// TwinCAT 3 PLC project Untitled1
// ProgramVersion: 3.1.4022.2
// libraries:
//   Tc2_MC2, * (Beckhoff Automation GmbH)
//   Tc2_NC, * (Beckhoff Automation GmbH)
//   Tc2_Standard, * (Beckhoff Automation GmbH)
//   Tc2_System, * (Beckhoff Automation GmbH)
//   Tc3_Module, * (Beckhoff Automation GmbH)
// project tree:
//   GVLs/ Global_Variables.TcGVL
//   / PlcTask.TcTTO
//   POUs/ FB_TcJoy.TcPOU, MAIN.TcPOU
//   POUs/Functions/ MAP.TcPOU
// real-time tasks:
//   TASK PlcTask: cycle T#10ms, priority 20, ADS port 350
// motion (NC):
//   TASK NC-Task 1 SAF: cycle T#2ms, priority 4, ADS port 501
//   TASK NC-Task 1 SVB: cycle T#10ms, priority 8, ADS port 511
//   AXIS Axis 1 (id 1)
//     Dynamic: Acceleration=7107.71, Deceleration=7107.71, Jerk=21323.1
//     Velo: RefSearch=47.3847210666667, RefSync=47.3847210666667, SlowManual=236.923605333333, FastManual=1421.541632, Fast=4738.47210666667, Maximum=4738.47
//     OtherSettings: AllowMotionCmdToSlave=true
//     encoder EncType=8
//       EncPara: ScaleFactorNumerator=104.8576, ScaleFactorDenominator=1048576, MaxCount=#xffffffff
//     drive DrvType=9
//       DrvPara: MaxCount=#xffffffff, DriveControlDWord=#x00030100
//         Analog: VeloReferenz=5212.31931733333, VeloScale=1.02400649589962, ScaleFactorActTorque=0.1
//         TimeComp: TaskDelayCycles=1
//     controller CtrType=1
//       CtrPara: PriorControlFactor=1
//         Observer: BandWidth=20
//   AXIS Axis B (id 2)
//     Dynamic: Acceleration=4539.33952, Deceleration=4539.33952, Jerk=13618.01856
//     Velo: RefSearch=30.2622634666667, RefSync=30.2622634666667, SlowManual=151.311317333333, FastManual=907.867904, Fast=3026.22634666667, Maximum=3026.22634666667
//     OtherSettings: AllowMotionCmdToSlave=true
//     encoder EncType=8
//       EncPara: ScaleFactorNumerator=104.8576, ScaleFactorDenominator=1048576, MaxCount=#xffffffff
//     drive DrvType=9
//       DrvPara: MaxCount=#xffffffff, DriveControlDWord=#x00030100
//         Analog: VeloReferenz=3328.84898133333, VeloScale=1.02400649589962, ScaleFactorActTorque=0.1
//         TimeComp: TaskDelayCycles=1
//     controller CtrType=1
//       CtrPara: PriorControlFactor=1
//         Observer: BandWidth=20
//   AXIS Axis 3 (id 3)
//     OtherSettings: AllowMotionCmdToSlave=true
//     encoder EncType=19
//       EncPara: MaxCount=#xffffffff
//     drive DrvType=16
//       DrvPara: MaxCount=#xffffffff
//         Analog: ScaleFactorActTorque=0.1
//         TimeComp: TaskDelayCycles=1
//     controller CtrType=1
//       CtrPara: PriorControlFactor=1
//         Observer: BandWidth=20
//   AXIS Axis 4 (id 4)
//     Dynamic: Acceleration=167
//     Velo: Maximum=720
//     OtherSettings: AllowMotionCmdToSlave=true
//     encoder EncType=1
//       EncPara: ScaleFactorNumerator=0.005625, Inverse=true
//         Inc: RefSearchInverse=true, RefSyncInverse=false, RefSoftSyncMask=#x0000ffff
//     drive DrvType=24
//       DrvPara: Inverse=true
//         Analog: VeloReferenz=720, ScaleFactorActTorque=0.1
//         TimeComp: TaskDelayCycles=1
//     controller CtrType=1
//       CtrPara: PriorControlFactor=1
//         Observer: BandWidth=20
// I/O:
//   DEVICE Local NIC (EtherCAT), AmsNetId 5.32.241.178.2.1
//     Drive 7 (AX5203-0000-0210) [AX5203-0000-0210 EtherCAT Drive (SoE, 2 Ch.)]
//     Term 1 (EK1100) [EK1100 EtherCAT Coupler (2A E-Bus)]
//       Term 2 (EL3255) [EL3255 5Ch. potentiometer measurement with sensor supply]
//       Term 3 (EL1008) [EL1008 8Ch. Dig. Input 24V, 3ms]
//       Term 4 (EL2008) [EL2008 8Ch. Dig. Output 24V, 0.5A]
//       Term 6 (EL9011) [EL9011 End Terminal]
//     Box 5 (EP2318-0001) [EP2318-0001 4 Ch. Dig. In, 10µs, 4 Ch. Dig. Out 24V, 0,5A, M8]
//   DEVICE Device 2 (EtherCAT), AmsNetId 5.32.241.178.3.1
//     Term 1 (EK1200) [EK1200-5000 EtherCAT Power supply (2A E-Bus)]
//       Term 9 (EL7201-0010) [EL7201-0010 1Ch. MDP742 Servo motor output stage with OCT (50V, 4A)]
//       Term 10 (EL7041) [EL7041 1Ch. Stepper motor output stage (50V, 5A)]
//       Term 4 (EL9011) [EL9011 End Terminal]
// variable links:
//   NC-Task 1 SAF/Axes/Axis 1 <-> Local NIC (EtherCAT)/Drive 7 (AX5203-0000-0210)
//     Drive/Inputs/In/nDataIn1 <-> AT 1/Following distance
//     Drive/Inputs/In/nDcOutputTime <-> InfoData/DcOutputShift
//     Drive/Inputs/In/nState1 <-> AT 1/Drive status word @bit 8
//     Drive/Inputs/In/nState2 <-> AT 1/Drive status word
//     Drive/Inputs/In/nState4 @bit 1 <-> WcState/InputToggle
//     Drive/Inputs/In/nState4 <-> WcState/WcState
//     Drive/Outputs/Out/nCtrl1 <-> MDT 1/Master control word @bit 8
//     Drive/Outputs/Out/nDataOut1 <-> MDT 1/Position command value
//     Enc/Inputs/In/nDataIn1 <-> AT 1/Position feedback 1 value
//     Enc/Inputs/In/nDcInputTime <-> InfoData/DcInputShift
//     Enc/Inputs/In/nState4 @bit 1 <-> WcState/InputToggle
//     Enc/Inputs/In/nState4 <-> WcState/WcState
//   NC-Task 1 SAF/Axes/Axis 3 <-> Device 2 (EtherCAT)/Term 1 (EK1200)/Term 9 (EL7201-0010)
//     Drive/Inputs/In/nDcOutputTime <-> InfoData/DcOutputShift
//     Drive/Inputs/In/nState1 <-> DRV Statusword/Statusword
//     Drive/Inputs/In/nState2 <-> DRV Statusword/Statusword @bit 8
//     Drive/Inputs/In/nState4 @bit 1 <-> WcState/InputToggle
//     Drive/Inputs/In/nState4 <-> WcState/WcState
//     Drive/Outputs/Out/nCtrl1 <-> DRV Controlword/Controlword
//     Drive/Outputs/Out/nCtrl2 <-> DRV Controlword/Controlword @bit 8
//     Drive/Outputs/Out/nDataOut2 <-> DRV Target velocity/Target velocity
//     Enc/Inputs/In/nDataIn1 <-> FB Position/Position
//     Enc/Inputs/In/nDcInputTime <-> InfoData/DcInputShift
//     Enc/Inputs/In/nState4 @bit 1 <-> WcState/InputToggle
//     Enc/Inputs/In/nState4 <-> WcState/WcState
//   NC-Task 1 SAF/Axes/Axis 4 <-> Device 2 (EtherCAT)/Term 1 (EK1200)/Term 10 (EL7041)
//     Drive/Inputs/In/nState1 @bit 3 <-> STM Status/Status/Error
//     Drive/Inputs/In/nState1 @bit 5 <-> STM Status/Status/Moving negative
//     Drive/Inputs/In/nState1 @bit 4 <-> STM Status/Status/Moving positive
//     Drive/Inputs/In/nState1 @bit 1 <-> STM Status/Status/Ready
//     Drive/Inputs/In/nState1 <-> STM Status/Status/Ready to enable
//     Drive/Inputs/In/nState1 @bit 6 <-> STM Status/Status/Torque reduced
//     Drive/Inputs/In/nState1 @bit 2 <-> STM Status/Status/Warning
//     Drive/Inputs/In/nState2 @bit 3 <-> STM Status/Status/Digital input 1
//     Drive/Inputs/In/nState2 @bit 4 <-> STM Status/Status/Digital input 2
//     Drive/Inputs/In/nState2 @bit 5 <-> STM Status/Status/Sync error
//     Drive/Inputs/In/nState2 @bit 7 <-> STM Status/Status/TxPDO Toggle
//     Drive/Inputs/In/nState4 @bit 1 <-> WcState/InputToggle
//     Drive/Inputs/In/nState4 <-> WcState/WcState
//     Drive/Outputs/Out/nCtrl1 <-> STM Control/Control/Enable
//     Drive/Outputs/Out/nCtrl1 @bit 2 <-> STM Control/Control/Reduce torque
//     Drive/Outputs/Out/nCtrl1 @bit 1 <-> STM Control/Control/Reset
//     Drive/Outputs/Out/nDataOut2[0] <-> STM Velocity/Velocity
//     Enc/Inputs/In/nDataIn1[0] <-> ENC Status compact/Counter value
//     Enc/Inputs/In/nDataIn2[0] <-> ENC Status compact/Latch value
//     Enc/Inputs/In/nState1 @bit 4 <-> ENC Status compact/Status/Counter overflow
//     Enc/Inputs/In/nState1 @bit 3 <-> ENC Status compact/Status/Counter underflow
//     Enc/Inputs/In/nState1 @bit 7 <-> ENC Status compact/Status/Extrapolation stall
//     Enc/Inputs/In/nState1 <-> ENC Status compact/Status/Latch C valid
//     Enc/Inputs/In/nState1 @bit 1 <-> ENC Status compact/Status/Latch extern valid
//     Enc/Inputs/In/nState1 @bit 2 <-> ENC Status compact/Status/Set counter done
//     Enc/Inputs/In/nState2 @bit 4 <-> ENC Status compact/Status/Status of extern latch
//     Enc/Inputs/In/nState2 <-> ENC Status compact/Status/Status of input A
//     Enc/Inputs/In/nState2 @bit 1 <-> ENC Status compact/Status/Status of input B
//     Enc/Inputs/In/nState2 @bit 2 <-> ENC Status compact/Status/Status of input C
//     Enc/Inputs/In/nState2 @bit 5 <-> ENC Status compact/Status/Sync error
//     Enc/Inputs/In/nState2 @bit 7 <-> ENC Status compact/Status/TxPDO Toggle
//     Enc/Inputs/In/nState4 @bit 1 <-> WcState/InputToggle
//     Enc/Inputs/In/nState4 <-> WcState/WcState
//     Enc/Outputs/Out/nCtrl1 <-> ENC Control compact/Control/Enable latch C
//     Enc/Outputs/Out/nCtrl1 @bit 3 <-> ENC Control compact/Control/Enable latch extern on negative edge
//     Enc/Outputs/Out/nCtrl1 @bit 1 <-> ENC Control compact/Control/Enable latch extern on positive edge
//     Enc/Outputs/Out/nCtrl1 @bit 2 <-> ENC Control compact/Control/Set counter
//     Enc/Outputs/Out/nDataOut1[0] <-> ENC Control compact/Set counter value
//   NC-Task 1 SAF/Axes/Axis B <-> Local NIC (EtherCAT)/Drive 7 (AX5203-0000-0210)
//     Drive/Inputs/In/nDataIn1 <-> AT 2/Following distance
//     Drive/Inputs/In/nDcOutputTime <-> InfoData/DcOutputShift
//     Drive/Inputs/In/nState1 <-> AT 2/Drive status word @bit 8
//     Drive/Inputs/In/nState2 <-> AT 2/Drive status word
//     Drive/Inputs/In/nState4 @bit 1 <-> WcState/InputToggle
//     Drive/Inputs/In/nState4 <-> WcState/WcState
//     Drive/Outputs/Out/nCtrl1 <-> MDT 2/Master control word @bit 8
//     Drive/Outputs/Out/nDataOut1 <-> MDT 2/Position command value
//     Enc/Inputs/In/nDataIn1 <-> AT 2/Position feedback 1 value
//     Enc/Inputs/In/nDcInputTime <-> InfoData/DcInputShift
//     Enc/Inputs/In/nState4 @bit 1 <-> WcState/InputToggle
//     Enc/Inputs/In/nState4 <-> WcState/WcState
//   Untitled1/Untitled1 Instance <-> Local NIC (EtherCAT)/Term 1 (EK1100)/Term 2 (EL3255)
//     PlcTask Inputs/MAIN.Throttle <-> AI Standard Channel 1/Value
//   Untitled1/Untitled1 Instance <-> Local NIC (EtherCAT)/Term 1 (EK1100)/Term 3 (EL1008)
//     PlcTask Inputs/MAIN.prox <-> Channel 5/Input
//   Untitled1/Untitled1 Instance <-> Local NIC (EtherCAT)/Term 1 (EK1100)/Term 4 (EL2008)
//     PlcTask Outputs/MAIN.four <-> Channel 4/Output
//     PlcTask Outputs/MAIN.one <-> Channel 1/Output
//     PlcTask Outputs/MAIN.three <-> Channel 3/Output
//     PlcTask Outputs/MAIN.two <-> Channel 2/Output
//   Untitled1/Untitled1 Instance <-> NC-Task 1 SAF/Axes/Axis 4
//     PlcTask Inputs/MAIN.AxisB.NcToPlc <-> Outputs/ToPlc
//     PlcTask Outputs/MAIN.AxisB.PlcToNc <-> Inputs/FromPlc

CONFIGURATION Untitled1
    RESOURCE PLC ON TwinCAT3
        TASK PlcTask(INTERVAL := T#10ms, PRIORITY := 20);
        PROGRAM MAIN WITH PlcTask : MAIN;
    END_RESOURCE
END_CONFIGURATION

// ---- GVLs/Global_Variables.TcGVL
VAR_GLOBAL
	
END_VAR

// ---- POUs/MAIN.TcPOU
PROGRAM MAIN
VAR
	
    heartbeat : BYTE;
	
	// Outputs.
	one AT %Q* : BOOL;
	two AT %Q* : BOOL;
	three AT %Q* : BOOL;
	four AT %Q* : BOOL;
	
	prox AT %I* : BOOL;  // Input
	
	// Dynamic Throttle
	Throttle AT %I* : INT;
	LastThrottle : INT;
	
	AxisB : AXIS_REF;

	McPower : MC_Power;
	McReset : MC_Reset;
	McJogging : MC_Jog;
	McVelocity : MC_MoveVelocity;
	McStop : MC_Stop;
	McHome : MC_Home;

	
    CurrentVelocityCmd : DINT;

	iState : DINT; // My State

	McMoveAbs : MC_MoveAbsolute;
	McMoveRel : MC_MoveRelative;
	iNumMoves : DINT:= 5;
	iCurrMove : DINT;
	fMoveDistEachTime : REAL:= 10;
	fRelMoveDist : REAL;
	
	TcJoy : FB_TcJoy;

END_VAR

heartbeat := heartbeat + 1;

CurrentVelocityCmd := MAP(Throttle,29800,22600,0,2800);
IF CurrentVelocityCmd < 50 THEN
	CurrentVelocityCmd := 0;
END_IF

AxisB.ReadStatus();

McPower(Axis:=AxisB,Enable:=TRUE,Enable_Positive:=TRUE,Enable_Negative:=TRUE);
McReset(Axis:=AxisB);
McJogging(Axis:=AxisB);
McHome(Axis:=AxisB,bCalibrationCam := prox);

McMoveAbs(Axis:=AxisB);
McMoveRel(Axis:=AxisB);

TcJoy();

CASE iState OF
	
    0:  // Initial

		iState := 10;

    10:  // Start Drive Reset

		McHome(Axis:=AxisB,Execute:=FALSE);
		McReset(Axis:=AxisB,Execute:=TRUE);
		IF McReset.Done THEN
			iState :=20;
		ELSIF McReset.Error THEN
			iState := 999;
		END_IF

    20:  // Wait for Drive to Reset

		IF McPower.Status AND (CurrentVelocityCmd > 1000 OR TcJoy.Y_Button) THEN
			iState := 100;
		END_IF	
		
    30:  // Wait for drive JOG command.
    
		IF TcJoy.iRightTrigger_Axis > 0 THEN
	
			IF TcJoy.iRightStick_X_Axis > 0 THEN
				McJogging.JogForward := TRUE;
				McJogging.Velocity := ABS(MAP(TcJoy.iRightStick_X_Axis,6000,32767,0,720));
			ELSE
				McJogging.JogForward := FALSE;
			END_IF
			IF TcJoy.iRightStick_X_Axis < 0 THEN
				McJogging.JogBackwards := TRUE;
				McJogging.Velocity := ABS(MAP(TcJoy.iRightStick_X_Axis,-6000,-32767,0,720));				
			ELSE
				McJogging.JogBackwards := FALSE;
			END_IF
			IF TcJoy.iRightStick_X_Axis = 0 THEN
				McJogging.JogForward := FALSE;
				McJogging.JogBackwards := FALSE;
			END_IF
			
			McJogging.Mode := MC_JOGMODE_CONTINOUS;
			McJogging.Acceleration := 500;
			McJogging.Deceleration := 500;
			McJogging.Jerk := 1000000;
			McJogging(Axis:=AxisB);
			
		ELSE
			McJogging.JogForward := FALSE;
			McJogging.JogBackwards := FALSE;
			iState := 200;
		END_IF 
		
	40:  // Wait for velocity command.
	
	//	McVelocity(Axis:=AxisB,
	//			Velocity:=CurrentVelocityCmd,
	///			Acceleration:=10000,
	//			Deceleration:=10000,
	//			Jerk:=1000000,
	//			Direction:=MC_Direction.MC_Positive_Direction,
	//			Execute:=prox AND (LastThrottle<>Throttle));
	//	IF NOT prox THEN
	//		McVelocity(Axis:=AxisB,Execute:=FALSE);
	//		iState := 900;
	//	END_IF				
	//	
		
		IF TcJoy.iLeftTrigger_Axis > 0 THEN
			
			McStop(Axis:=AxisB,Execute:=FALSE);
			
			IF TcJoy.iRightStick_X_Axis > 0 THEN
				McVelocity.Velocity := ABS(MAP(TcJoy.iRightStick_X_Axis,6000,32767,0,720));
			END_IF
			IF TcJoy.iRightStick_X_Axis < 0 THEN
				McVelocity.Velocity := ABS(MAP(TcJoy.iRightStick_X_Axis,-6000,-32767,0,720));				
			END_IF
			IF TcJoy.iRightStick_X_Axis = 0 THEN
				McVelocity.Velocity := 0;
			END_IF

			McVelocity(Axis:=AxisB, Execute:=LastThrottle<>Throttle);
			
		ELSE
			McVelocity(Axis:=AxisB, Execute:=FALSE);
			McStop(Axis:=AxisB,Execute:=TRUE);
			iState := 200;
		END_IF 
		
		LastThrottle:=Throttle;
		
	100:  // Start Homing Process.
		
		McHome(Axis:=AxisB,bCalibrationCam:=prox,Execute:=TRUE);
		IF McHome.Busy THEN
			iState := 110;
		END_IF
		
	110: // Homing running, wait for homing to complete.
	
		IF McHome.Done AND NOT McHome.Error THEN
			McHome(Axis:=AxisB,Execute:=FALSE);
			iState := 200;
		ELSIF McHome.Error THEN
			McHome(Axis:=AxisB,Execute:=FALSE);
			iState := 999;
		END_IF
		
	200: // Homing Complete.  Ready to Run.
		
		IF TcJoy.Y_Button THEN // Home
			iState := 100;	
		END_IF
		IF TcJoy.B_Button THEN // Run dance move
			iState := 300;
		END_IF
		IF TcJoy.iRightTrigger_Axis > 0 THEN // Jog with joystick
			iState := 30;
		END_IF
		IF TcJoy.iLeftTrigger_Axis > 0 THEN // ABS with joystick
			iState := 600;
		END_IF
		
 	300:  // Start ABS Move to center to prep for processing part
	
	    McMoveAbs(Axis:=AxisB,
					Position := 100,
					Velocity := 100,
					Acceleration := 500,
					Deceleration := 500,
					Jerk := 100000,
					Execute:=TRUE);
					
		iState := 310;
		
	310:  // Wait for abs move to complete.
	
	    IF McMoveAbs.Done AND NOT McMoveAbs.Error THEN
			McMoveAbs(Axis:=AxisB,Execute:=FALSE);
			iCurrMove := 1;
			iState := 400;
		ELSIF McMoveAbs.Error THEN
			McMoveAbs(Axis:=AxisB,Execute:=FALSE);
			iState := 999;	
		END_IF
		
	400:  // Start Rel Moves.
	
	    // More to do?
		IF iCurrMove < iNumMoves THEN
			// increment move counter for next time.
			iCurrMove := iCurrMove + 1;
			// Calculate Distance
			fRelMoveDist := DINT_TO_REAL(iCurrMove) * fMoveDistEachTime;
			iState := 410;
		ELSE
			// Nothing to do.
			iState := 500;
		END_IF
		
	410:  // Start rel move in pos direction
		
	    McMoveRel(Axis:=AxisB,
					Distance := fRelMoveDist,
					Velocity := 720,
					Acceleration := 2000,
					Deceleration := 2000,
					Jerk := 1000000,
					Execute:=TRUE);
					
		iState := 420;
		
	420:  // Wait on rel move to complete
	
		IF McMoveRel.Done AND NOT McMoveRel.Error THEN
			McMoveRel(Axis:=AxisB,Execute:=FALSE);
			iState := 450;
		ELSIF McMoveRel.Error THEN
			McMoveRel(Axis:=AxisB,Execute:=FALSE);
			iState := 999;	
		END_IF
		
	450:  // Move negative rel back to start position
					
		McMoveRel(Axis:=AxisB,
					Distance := -fRelMoveDist,
					Velocity := 720,
					Acceleration := 2000,
					Deceleration := 2000,
					Jerk := 1000000,
					Execute:=TRUE);
					
		iState := 460;
		
	460:  // Wait on rel move to complete
	
		IF McMoveRel.Done AND NOT McMoveRel.Error THEN
			McMoveRel(Axis:=AxisB,Execute:=FALSE);
			iState := 400;
		ELSIF McMoveRel.Error THEN
			McMoveRel(Axis:=AxisB,Execute:=FALSE);
			iState := 999;	
		END_IF

	500:  // Start ABS Move Back to home
	
	    McMoveAbs(Axis:=AxisB,
					Position := 0,
					Velocity := 100,
					Acceleration := 100,
					Deceleration := 100,
					Jerk := 100000,
					Execute:=TRUE);
					
		iState := 510;
		
	510:  // Wait for abs move to complete.
	
	    IF McMoveAbs.Done AND NOT McMoveAbs.Error THEN
			McMoveAbs(Axis:=AxisB,Execute:=FALSE);
			iCurrMove := 1;
			iState := 200;
		ELSIF McMoveAbs.Error THEN
			McMoveAbs(Axis:=AxisB,Execute:=FALSE);
			iState := 999;	
		END_IF		
		
		
	600:   // Start ABS Move from joystick
	
		IF TcJoy.iLeftTrigger_Axis > 0 THEN
	
			IF TcJoy.iRightStick_X_Axis > 0 THEN
				McMoveAbs.Position := ABS(MAP(TcJoy.iRightStick_X_Axis,6000,32767,100,200));
			END_IF
			IF TcJoy.iRightStick_X_Axis < 0 THEN
				McMoveAbs.Position := ABS(MAP(TcJoy.iRightStick_X_Axis,-32767,-6000,0,100));				
			END_IF
			IF TcJoy.iRightStick_X_Axis = 0 THEN
				McMoveAbs.Position := 100;
			END_IF

			McMoveAbs(Axis:=AxisB,
					Velocity := 500,
					Acceleration := 500,
					Deceleration := 2000,
					Jerk := 1000000,
					Execute:=TRUE);
					
			iState := 610;
			
		ELSE
			McMoveAbs(Axis:=AxisB,Execute:=FALSE);
			iState := 200;
		END_IF 
	

		
	610:  // Wait for abs move to complete.
	
	    IF McMoveAbs.Done AND NOT McMoveAbs.Error THEN
			McMoveAbs(Axis:=AxisB,Execute:=FALSE);
			iState := 600;
		ELSIF McMoveAbs.Error THEN
			McMoveAbs(Axis:=AxisB,Execute:=FALSE);
			iState := 999;	
		END_IF	
	
	900:  // Stop servo.
	
	    McStop(Axis:=AxisB,Execute:=TRUE);
		IF prox THEN
			McStop(Axis:=AxisB,Execute:=FALSE);
			iState := 40;
		END_IF
	
	999: // Handle Error (TODO)

END_CASE

END_PROGRAM

// ---- POUs/FB_TcJoy.TcPOU
FUNCTION_BLOCK FB_TcJoy
VAR_INPUT
END_VAR
VAR_OUTPUT
	bIsActive : BOOL;  // Are we running?
	// Controller Outputs for use in programs:
	Start_Button : BOOL; 
	Back_Button : BOOL;
	A_Button : BOOL;
	B_Button : BOOL;
	X_Button : BOOL;
	Y_Button : BOOL;
	LeftShoulder_Button : BOOL;
	RightShoulder_Button : BOOL;
	LeftStick_Button : BOOL;
	RightStick_Button : BOOL;
	DPad_Up_Button : BOOL;
	DPad_Left_Button : BOOL;
	DPad_Right_Button : BOOL;
	DPad_Down_Button : BOOL;
	iLeftStick_X_Axis : DINT;
	iLeftStick_Y_Axis : DINT;
	iRightStick_X_Axis : DINT;
	iRightStick_Y_Axis : DINT;
	iLeftTrigger_Axis : DINT;
	iRightTrigger_Axis  : DINT;
	sBatteryInfo		: STRING;
END_VAR
VAR
	// From VB App To PLC
	bHeartBeatToggle : BOOL;  // From VB App
	iADSWatchdogMS : DINT;    // If Rate is > this, all outputs go to 0.
	iADSWatchdogDeadDurationMS : DINT;    // If watchdog trips, outputs go to 0 for this long.
	bWatchdogFailureActive			: BOOL;
	// From PLC To VB (Status)
	iUpdateRateMS : DINT;    // Rate in MS between heartbeat changes detected.
	
	// Internal Use Only
	HeartBeatChanged_RTRIG : R_TRIG;
	bHeartBeatToggle_Last : BOOL;
	UpdateRate_TMR : TON;
	
	LatencyWatchdog_TMR : TON; // Watch for missing ADS and kill joy output for a while.
	LatencyWatchdogDeadDuration_TMR : TON; // Watchdog will kill the outputs for this long...
	
	iScanCount: DINT; // Scan counter for VB Status.
	
	bControllerConnected : BOOL;  // Is there a controller connected?
	
END_VAR


// NOTE: This code is intended to run with TcJoy, an as-of-now closed source .NET application that talks to xbox 360 controllers and publishes the data over ADS to TwinCAT. 
// Email Evanmj@gmail.com for more info.

iScanCount := iScanCount+1;

UpdateRate_TMR(PT:=T#999M);

HeartBeatChanged_RTRIG(clk := bHeartBeatToggle <> bHeartBeatToggle_Last);

// VB "Just" changed heartbeat.
IF HeartBeatChanged_RTRIG.Q THEN
	bHeartBeatToggle_Last := bHeartBeatToggle;
	iUpdateRateMS := TIME_TO_DINT(UpdateRate_TMR.ET); // Grab Elapsed Time
	UpdateRate_TMR(IN:=FALSE); // Reset Timer
	UpdateRate_TMR(IN:=TRUE); // Reset Timer
END_IF

LatencyWatchdog_TMR(IN:=bHeartBeatToggle, PT:=DINT_TO_TIME(iADSWatchdogMS));

// AHH Latency Elapsed!
IF LatencyWatchdog_TMR.Q THEN
	bWatchdogFailureActive := TRUE;
	bControllerConnected := FALSE;
END_IF

LatencyWatchdogDeadDuration_TMR(IN:=bWatchdogFailureActive, PT:=DINT_TO_TIME(iADSWatchdogDeadDurationMS));

// ReEnable after setting duration expires
IF LatencyWatchdogDeadDuration_TMR.Q THEN
	bWatchdogFailureActive := FALSE;
END_IF

// Null the outputs on WD Active so we don't jog into a wall if we lose connection.
IF bWatchdogFailureActive OR NOT bControllerConnected THEN
	Start_Button := FALSE; 
	Back_Button := FALSE; 
	A_Button := FALSE; 
	B_Button := FALSE; 
	X_Button := FALSE; 
	Y_Button := FALSE; 
	LeftShoulder_Button := FALSE; 
	RightShoulder_Button := FALSE; 
	LeftStick_Button := FALSE; 
	RightStick_Button := FALSE; 
	DPad_Up_Button := FALSE; 
	DPad_Left_Button := FALSE; 
	DPad_Right_Button := FALSE; 
	DPad_Down_Button := FALSE; 
	iLeftStick_X_Axis := 0;
	iLeftStick_Y_Axis := 0;
	iRightStick_X_Axis := 0;
	iRightStick_Y_Axis := 0;
	iLeftTrigger_Axis := 0;
	iRightTrigger_Axis := 0;
	sBatteryInfo		:= 'Unkn';
	
	UpdateRate_TMR(IN:=FALSE); // Reset Rate Timer
ELSE
	; // All is well, VB will update our values constantly.
END_IF

bIsActive := NOT bWatchdogFailureActive AND bControllerConnected;

END_FUNCTION_BLOCK

// ---- POUs/Functions/MAP.TcPOU
// Just like arduino 'Map".  Rescales.  Evanmj@gmail.com
FUNCTION MAP : DINT
VAR_INPUT
	x : DINT;
	in_min : DINT;
	in_max : DINT;
	out_min : DINT;
	out_max : DINT;
	
END_VAR
VAR
END_VAR


IF ((in_max - in_min) + out_min) <> 0 THEN
	MAP := DINT_TO_INT((x - in_min) * (out_max - out_min) / (in_max - in_min) + out_min);
ELSE
	MAP := 0;
END_IF

RETURN;

END_FUNCTION
